PROGRAM MAIN
VAR

END_VAR

superimpose();

END_PROGRAM

(* stored: Version 1.1.0.1, ProductVersion 3.1.4024.4
   POU MAIN: Id {27ce5a08-4f57-4c86-8d17-7f73b57b23c2}, SpecialFunc None *)
